// Struckig
// Copyright (C) 2022 Stefan Besler

// This program is free software: you can redistribute it and/or modify
// it under the terms of the GNU General Public License as published by
// the Free Software Foundation, either version 3 of the License, or
// (at your option) any later version.

// This program is distributed in the hope that it will be useful,
// but WITHOUT ANY WARRANTY; without even the implied warranty of
// MERCHANTABILITY or FITNESS FOR A PARTICULAR PURPOSE.  See the
// GNU General Public License for more details.
//
// You should have received a copy of the GNU General Public License
// along with THIS PROGRAM.  IF NOT, see <http://www.gnu.org/licenses/>.
{attribute 'qualified_only'}
{attribute 'strict'}
/// Defines whether synchronized trajectory duration is continuous or cycle-discrete.
TYPE DiscretizationType :
(
  Continuous, //< Every synchronization duration is allowed.
  Discrete //< Synchronization duration must be a multiple of cycle time.
);
END_TYPE

(* stored: Version 1.1.0.1
   DUT DiscretizationType: Id {57780566-a3c2-481a-ac6d-a6d55abca32c} *)
